FUNCTION_BLOCK iCreateAdvButton (* LMS LED on Light Sensor *)
  (* Standard: 61499-2 *)
  (* Version 0.0, 2012-07-02, 4DIAC-IDE, 4DIAC-Consortium *)
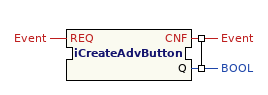
  EVENT_INPUT
    REQ; (* Service Request *)
  END_EVENT
  EVENT_OUTPUT
    CNF WITH Q; (* Confirmation of Requested Service *)
  END_EVENT
  VAR_OUTPUT
    Q : BOOL; (* True if Advance Button pressed *)
  END_VAR
  SERVICE APPLICATION/RESOURCE (* LMS LED on Light Sensor *)
    SEQUENCE normal_establishment
      APPLICATION.INIT+(PARAMS) -> APPLICATION.INITO+(PARAMS);
    END_SEQUENCE
    SEQUENCE unsuccessful_establishment
      APPLICATION.INIT+(PARAMS) -> APPLICATION.INITO-(STATUS);
    END_SEQUENCE
    SEQUENCE request_confirm
      APPLICATION.REQ+(SD) -> APPLICATION.CNF+(RD);
    END_SEQUENCE
    SEQUENCE request_inhibited
      APPLICATION.REQ-(SD) -> APPLICATION.CNF-(STATUS);
    END_SEQUENCE
    SEQUENCE request_error
      APPLICATION.REQ+(SD) -> APPLICATION.CNF-(STATUS);
    END_SEQUENCE
    SEQUENCE indication_response
      RESOURCE.indicate(RD) -> APPLICATION.IND+(RD);
      APPLICATION.RSP(QI,SD) -> RESOURCE.response(QI,SD);
    END_SEQUENCE
    SEQUENCE indication_inhibited
      RESOURCE.indicate(RD,QI=FALSE) -> RESOURCE.inhibited();
    END_SEQUENCE
    SEQUENCE error_indication
      RESOURCE.error(STATUS) -> APPLICATION.IND-(STATUS);
    END_SEQUENCE
    SEQUENCE application_initiated_termination
      APPLICATION.INIT-() -> APPLICATION.INITO-(STATUS);
    END_SEQUENCE
    SEQUENCE resource_initiated_termination
      -> APPLICATION.INITO-(STATUS);
    END_SEQUENCE
  END_SERVICE
END_FUNCTION_BLOCK
